# EPICS substitutions: db/Beckhoff_6XXX/ecmcEL6022.substitutions
file "ecmcEcSlave.template"
{
  pattern {}
          {}
}

file "ecmcEL60X2-chX.template"
{
  pattern {CH_ID, NELM }
          {01,     22   }
          {02,     22   }
}
